{attribute addProperty BoxType "ELX1054-0000-0016"}
{attribute addProperty Id "ChannelAT %I*ARRAY[0..3] OF Channel_E18390666480Input_Type_NCAT %I*Input_Type_NC_3EE6969D3240WcStateAT %I*WcState_F855686C1620InfoDataAT %I*InfoData_192954DE1620"}
{attribute addProperty CRC "715122290"}
{attribute addProperty SizeInBites "128"}
{attribute addProperty SizeInBytes "16"}
TYPE ELX1054_FE7182BE :
STRUCT
	{attribute addProperty Name "Channel"}
	Channel : ARRAY[0..3] OF Channel_E1839066;
	{attribute addProperty Name "Input_Type_NC"}
	Input_Type_NC : Input_Type_NC_3EE6969D;
	{attribute addProperty Name "WcState"}
	WcState : WcState_F855686C;
	{attribute addProperty Name "InfoData"}
	InfoData : InfoData_192954DE;
END_STRUCT
END_TYPE

(* stored: Version 1.2.0.0, ProductVersion 3.1.4024.9
   DUT ELX1054_FE7182BE: Id {f37b50c5-5179-443d-ba3b-c51fffe80e65} *)
